(* Logix 5000 project; controller AdvManLab vendor 1 type 14 code 158 rev 28.12; software revision 28.01; part 4 of 13 *)
(* tags used below, declared in another part *)
   Inp : P_PF52x_Inp;   // Common part of PF523 / PF525 Input Assembly
   Out : P_PF52x_Out;   // Common part of PF523 / PF525 Output Assembly
   Inp_FwdPermOK : BOOL;   // 1=Permissives OK, drive can start Forward
   Inp_FwdNBPermOK : BOOL;   // 1=Non-Bypassable Permissives OK, drive can start Forward
   Inp_RevPermOK : BOOL;   // 1=Permissives OK, drive can start Reverse
   Inp_RevNBPermOK : BOOL;   // 1=Non-Bypassable Permissives OK, motor can start Reverse
   Inp_IntlkOK : BOOL;   // 1=Interlocks OK, drive can start/run
   Inp_NBIntlkOK : BOOL;   // 1=Non-Bypassable Interlocks OK, drive can start/run
   Inp_IOFault : BOOL;   // Input Communication Status 0=OK, 1=fail
   Inp_Sim : BOOL;   // 1=Simulate working drive; 0=Start/Stop/ Monitor actual drive
   Inp_Hand : BOOL;   // 1=Acquire Hand (typ. hardwired local) Mode, 0=Release Hand Mode
   Inp_OvrdCmd : SINT;   // Override Mode Command: 0=None, 1=Stop, 2=Start Fwd 3=Start Rev
   Inp_OvrdSpeed : REAL;   // Value to set Speed Reference in Override Mode (SpeedRef EU)
   Inp_Reset : BOOL;   // 1=Reset drive fault conditions and latched Alarms
   Cfg_HasReverse : BOOL;   // 1=Drive can be run reverse, 0=Forward only
   Cfg_AllowLocal : BOOL;   // 1=Allow Local Start/Stop without alarm, 0=Start/Stop from HMI/prog only
   Cfg_SetTrack : BOOL;   // 1=PSets track OSets in Oper, OSets track PSets in Prog, 0=no tracking
   Cfg_SetTrackOvrdHand : BOOL;   // 1=Prog/Oper Settings track Override/Hand speed reference
   Cfg_PCmdClear : ALIAS FOR Mode.Cfg_PCmdClear;
   Cfg_OCmdResets : BOOL;   // 1=New Oper drive cmd. resets fault, 0=reset req'd to clear fault
   Cfg_OvrdPermIntlk : BOOL;   // 1=Override ignores Bypassable Perm/ Intlk; 0=always use Perm/Intlk
   Cfg_ShedOnIOFault : BOOL;   // 1=Stop Motor and Alarm on I/O Fault; 0=Alarm only on I/O Fault
   Cfg_SimScaleEU : BOOL;   // 1=In simulation, scale Speed Ref EU to Speed Fdbk EU
   Cfg_SimScaleRaw : BOOL;   // 1=In simulation, scale Speed Ref EU to raw, then raw to Speed Fdbk EU
   Cfg_MinSpdRef : REAL;   // Minimum Speed Reference in EU (for limiting)
   Cfg_MaxSpdRef : REAL;   // Maximum Speed Reference in EU (for limiting)
   Cfg_SpeedRefRawMin : INT;   // Speed Reference Minimum in Drive (raw) Units (for scaling)
   Cfg_SpeedRefRawMax : INT;   // Speed Reference Maximum in Drive (raw) Units (for scaling)
   Cfg_SpeedRefEUMin : REAL;   // Speed Reference Minimum in Engineering Units (for scaling)
   Cfg_SpeedRefEUMax : REAL;   // Speed Reference Maximum in Engineering Units (for scaling)
   Cfg_SpeedFdbkRawMin : INT;   // Speed Feedback Minimum in Drive (raw) Units (for scaling)
   Cfg_SpeedFdbkRawMax : INT;   // Speed Feedback Maximum in Drive (raw) Units (for scaling)
   Cfg_SpeedFdbkEUMin : REAL;   // Speed Feedback Minimum in Engineering Units (for scaling)
   Cfg_SpeedFdbkEUMax : REAL;   // Speed Feedback Maximum in Engineering Units (for scaling)
   Cfg_SimRampT : DINT;   // Time to ramp speed fdbk when in Simulation (sec)
   Cfg_FailToStartT : DINT;   // Time after Start to get Run Feedback before Fault (sec)
   Cfg_FailToStopT : DINT;   // Time after Stop to drop Run Feedback before Fault (sec)
   Cfg_ResetPulseT : DINT;   // Time to pulse Out_Reset to clear drive fault
   Cfg_MaxJogT : REAL;   // Maximum jog time (sec, 0=unlimited)
   Cfg_OperKeep : SINT;   // Oper keeps control in Prog Mode: .0=Reference, .1=Start/Stop, .2=Fwd/Rev
   Cfg_ProgKeep : SINT;   // Prog keeps control in Oper Mode: .0=Reference, .1=Start/Stop, .2=Fwd/Rev
   PSet_SpeedRef : REAL;   // Program Setting of Speed Reference (EU)
   PSet_Owner : DINT;   // Program Owner Request ID (non-zero) or Release (zero)
   OSet_SpeedRef : REAL;   // Operator Setting of Speed Reference (EU)
   PCmd_Start : BOOL;   // Program Command to Start Drive
   PCmd_Fwd : BOOL;   // Program Command to set direction to Fowrard
   PCmd_Rev : BOOL;   // Program Command to set direction to Reverse
   PCmd_Reset : BOOL;   // Program Command to Reset drive fault and all Alarms requiring Reset
   PCmd_FailToStartAck : ALIAS FOR FailToStart.PCmd_Ack;   // Program Command to Acknowledge Fail to Start Alarm
   PCmd_FailToStopAck : ALIAS FOR FailToStop.PCmd_Ack;   // Program Command to Acknowledge Fail to Stop Alarm
   PCmd_IntlkTripAck : ALIAS FOR IntlkTrip.PCmd_Ack;   // Program Command to Acknowledge Interlock Trip Alarm
   PCmd_DriveFaultAck : ALIAS FOR DriveFault.PCmd_Ack;   // Program Command to Acknowledge Drive Fault Alarm
   PCmd_IOFaultAck : ALIAS FOR IOFault.PCmd_Ack;   // Program Command to Acknowledge I/O Fault Alarm
   OCmd_Start : BOOL;   // Operator Command to Start Drive
   OCmd_Stop : BOOL;   // Operator Command to Stop Drive
   OCmd_Jog : BOOL;   // Operator Command to Jog Drive (not cleared by P_PF52x!)
   OCmd_Fwd : BOOL;   // Operator Command to set direction to Forward
   OCmd_Rev : BOOL;   // Operator Command to set direction to Reverse
   OCmd_Bypass : BOOL;   // Operator Command to Bypass all Bypassable Interlocks and Permissives
   OCmd_Check : BOOL;   // Operator Command to Check (not bypass) all Interlocks and Permissives
   MCmd_Disable : BOOL;   // Maintenance Command to Disable Drive
   MCmd_Enable : BOOL;   // Maintenance Command to Enable (allow to run) Drive
   OCmd_Reset : BOOL;   // Operator Command to Reset all Alarms requiring Reset
   OCmd_ResetAckAll : BOOL;   // Operator Command to Reset all Alarms and latched Shed conditions
   Val_SpeedFdbk : REAL;   // Speed Feedback (actual) from drive
   Val_SpeedRefEUMin : REAL;   // Minimum of Speed Reference = MIN (Cfg_SpeedFdbkEUMin, Cfg_SpeedFdbkEUMax)
   Val_SpeedRefEUMax : REAL;   // Maximum of Speed Reference = MAX (Cfg_SpeedFdbkEUMin, Cfg_SpeedFdbkEUMax)
   Val_SpeedFdbkEUMin : REAL;   // Minimum of Speed Feedback = MIN (Cfg_SpeedFdbkEUMin, Cfg_SpeedFdbkEUMax)
   Val_SpeedFdbkEUMax : REAL;   // Maximum of Speed Feedback = MAX (Cfg_SpeedFdbkEUMin, Cfg_SpeedFdbkEUMax)
   Val_Fdbk : SINT;   // Device Feedback 0=Stopped, 1=Running Fwd 2=Running Rev 3=Accelerating 4=Decelerating
   Val_Owner : DINT;   // Current Object Owner ID (0=not owned)
   Sts_Starting : BOOL;   // 1=Drive requested to run and awaiting run feedback
   Sts_Running : BOOL;   // 1=Drive requested to run and is confirmed running
   Sts_CommandDir : BOOL;   // 1=Drive commanded to Forward, 0=Reverse
   Sts_ActualDir : BOOL;   // 1=Drive Actual direction is Forward, 0=Reverse
   Sts_Accel : BOOL;   // 1=Drive is Accelerating
   Sts_Decel : BOOL;   // 1=Drive is Decelerating
   Sts_NotReady : BOOL;   // 1=Device Not Ready, see detail bits for reason
   Sts_AtSpeed : BOOL;   // 1=Drive is running at reference speed
   Sts_Available : BOOL;   // 1=Drive available for control by automation (Prog)
   Sts_Bypass : BOOL;   // 1=Bypassable Interlocks and Permissives are Bypassed
   Sts_BypActive : BOOL;   // 1=Bypassing Active (Bypassed or Maintenance)
   Sts_Disabled : BOOL;   // 1=Drive is Disabled
   Sts_NotRdy : BOOL;   // 1=Motor is Not Ready to Run (independent of Mode)
   Nrdy_Disabled : BOOL;   // 1=Device Not Ready: Device Disabled by Maintenance
   Nrdy_CfgErr : BOOL;   // 1=Device Not Ready: Configuration Error
   Nrdy_Intlk : BOOL;   // 1=Device Not Ready: Interlock Not OK
   Nrdy_Perm : BOOL;   // 1=Device Not Ready: Permissive Not OK
   Nrdy_OperPrio : BOOL;   // 1=Device Not Ready: Operator State 0 Priority Command Requires Reset
   Nrdy_Fail : BOOL;   // 1=Device Not Ready: Device Failure (Shed Requires Reset)
   Nrdy_IOFault : BOOL;   // 1=Device Not Ready: I/O Fault (Shed Requires Reset)
   Nrdy_Trip : BOOL;   // 1=Device not Ready: Deivce Tripped (Drive Fault)
   Nrdy_DriveNR : BOOL;   // 1=Device Note Ready: Drive Not Ready
   Nrdy_NoMode : BOOL;   // 1=Device Not Ready: Device Logic Disabled / NO Mode
   Sts_MaintByp : BOOL;   // 1=A Maintenance Bypass is Active, display icon
   Sts_Err : BOOL;   // 1=Error in Config: see detail bits for reason
   Err_Timer : BOOL;   // 1=Error in Config: Invalid Check or Reset Pulse Time (use 0 to 2147483)
   Err_Sim : BOOL;   // 1=Error in Config: simulation timer preset: use 0 to 2147483)
   Err_Alarm : BOOL;   // 1=Error in Config: Alarm Min On Time, Shelf Time, Severity
   Err_FdbkRaw : BOOL;   // 1=Erron in Config: Speed Fdbk Raw Min = Max
   Err_FdbkEU : BOOL;   // 1=Error in Config: Speed Fdbk EU Min = Max
   Err_RefLim : BOOL;   // 1=Error in Config: Speed Ref Limit Min > Max
   Err_RefEU : BOOL;   // 1=Error in Config: Speed Ref EU Min = Max
   Err_RefRaw : BOOL;   // 1=Error in Config: Speed Ref Raw Min = Max
   Sts_Hand : ALIAS FOR Mode.Sts_Hand;
   Sts_Maint : ALIAS FOR Mode.Sts_Maint;
   Sts_Ovrd : ALIAS FOR Mode.Sts_Ovrd;
   Sts_Prog : ALIAS FOR Mode.Sts_Prog;
   Sts_Oper : ALIAS FOR Mode.Sts_Oper;
   Sts_FailToStart : ALIAS FOR FailToStart.Inp;   // 1=Drive Failed to Start (One-Shot)
   Sts_FailToStop : ALIAS FOR FailToStop.Inp;   // 1=Drive Failed to Stop
   Sts_IntlkTrip : ALIAS FOR IntlkTrip.Inp;   // 1=Drive was stopped by an Interlock NOT OK (One-Shot)
   Sts_DriveFault : ALIAS FOR DriveFault.Inp;   // 1=Drive Fault (see drive display or manual)
   Sts_IOFault : ALIAS FOR IOFault.Inp;   // I/O Comm Fault Status (0=OK, 1=Bad)
   Rdy_Fwd : BOOL;   // 1=Ready to receive OCmd_Fwd (enabled HMI button)
   Rdy_Rev : BOOL;   // 1=Ready to receive OCmd_Rev (enables HMI button)
   Rdy_Bypass : BOOL;   // 1=Ready to receive OCmd_Bypass (enables HMI button)
   Rdy_Check : BOOL;   // 1=Ready to receive OCmd_Check (enables HMI button)
   Rdy_Disable : BOOL;   // 1=Ready to receive MCmd_Disable (enables HMI button)
   Rdy_Enable : BOOL;   // 1=Ready to receive MCmd_Enable (enables HMI button)
   Rdy_SpeedRef : BOOL;   // 1=Ready to receive OSet_SpeedRef (enables data entry field)
   P_PF52x : BOOL;   // Unique Parameter Name for auto - discovery
   Mode : P_Mode;   // Drive Mode Selection
   IOFault : P_Alarm;   // I/O Fault Alarm
   IntlkTrip : P_Alarm;   // Interlock Trip Alarm
   FailToStop : P_Alarm;   // Drive Failed to Stop Alarm
   FailToStart : P_Alarm;   // Drive Failed to Start Alarm
   Cfg_Tag : STRING_20;   // Tagname for display on HMI
   Cfg_Label : STRING_20;   // Label for graphic symbol displayed on HMI
   Cfg_Desc : STRING_40;   // Description for display on HMI
   Wrk_Run : BOOL;   // 1=Drive should be "running", 0=should be "stopped"
   Wrk_StartRetrigT : TIMER;   // Time to pulse start output on start command retrigger (Maint)
   Wrk_StopRetrigT : TIMER;   // Time to pulse stop output on stop command retrigger (Maint)
   Wrk_RunFdbk : BOOL;   // Run Feedback based on mode, simulation, etc. 1=running
   Wrk_Bypass : BOOL;   // Internal Bypassable Permissives and Interlocks are Bypassed flag
   Wrk_Disabled : BOOL;   // Internal Drive is Disabled
   DriveFault : P_Alarm;   // Drive Faulted Alarm
   Cfg_SpeedRefEU : STRING_8;   // Speed Reference Engineering Units for display on HMI
   Wrk_SpeedRef : REAL;   // Working copy of Speed Reference (for limiting)
   Wrk_Rev : BOOL;   // Working (internal) Direction 1=Reverse 0=Forward (default)
   Wrk_Jog : BOOL;   // 1=Jog Drive, 0=Drive not jogging
   Wrk_ResetT : TIMER;   // Reset Output Pulse Timer
   Wrk_ResetONS : BOOL;   // One-Shot to fire Reset Timer to ensure min. output ON time.
   Cfg_SpeedFdbkEU : STRING_8;   // Speed Feedback Engineering Units for display on HMI
   Cfg_RevText : STRING_16;   // Name for Reverse Direction, e.g., "Down", "Reverse"
   Cfg_FwdText : STRING_16;   // Name for Forward Direction, e.g., "Up", "Forward"
   Wrk_StopT : TIMER;   // Stop Check Timer (for Fail to Stop)
   Wrk_StartT : TIMER;   // Start Check Timer (for Fail to Start)
   Wrk_Retrigger : BOOL;   // Maint Start issued while running or Stop while stopped
   Wrk_Step : REAL;   // Amount to change simulated Speed Fdbk this scan (ramp)
   Wrk_ScanTime : REAL;   // Seconds since previous scan
   Wrk_ScanT : TIMER;   // Scan Timer (milliseconds, always runs)
   Wrk_SimFdbkTgt : REAL;   // Speed Ref converted to Speed Fdbk units for simulation: target speed fdbk
   Inf_Type : STRING_16;   // Type identifier for HMI navigation
   Wrk_JogT : TIMER;   // Jog Timer
   Val_FaultDesc : STRING_40;   // Description of Drive Fault (given LastFaultCode)
   Wrk_ProgKeep2ONS : BOOL;   // Prog Keep bit 2 one-shot store
   Wrk_ProgKeep1ONS : BOOL;   // Prog Keep bit 1 one-shot store
   Wrk_ProgKeep0ONS : BOOL;   // Prog Keep bit 0 one-shot store
   Wrk_OperKeep2ONS : BOOL;   // Oper Keep bit 2 one-shot store
   Wrk_OperKeep1ONS : BOOL;   // Oper Keep bit 1 one-shot store
   Wrk_OperKeep0ONS : BOOL;   // Oper Keep bit 0 one-shot store
   Inf_Lib : STRING_12;   // Display Library for Faceplate call-up
   Cfg_DigIn4Txt : STRING_20;   // Drive Digital Input 4 Label
   Cfg_DigIn3Txt : STRING_20;   // Drive Digital Input 3 Label
   Cfg_DigIn2Txt : STRING_20;   // Drive Digital Input 2 Label
   Cfg_DigIn1Txt : STRING_20;   // Drive Digital Input 1 Label
   ONS : DINT;
   Running : BOOL;
(* P_PF52x, continued *)

ROUTINE Logic   (* ladder *)
// Normal Scan: control / monitor Variable-Speed Drive
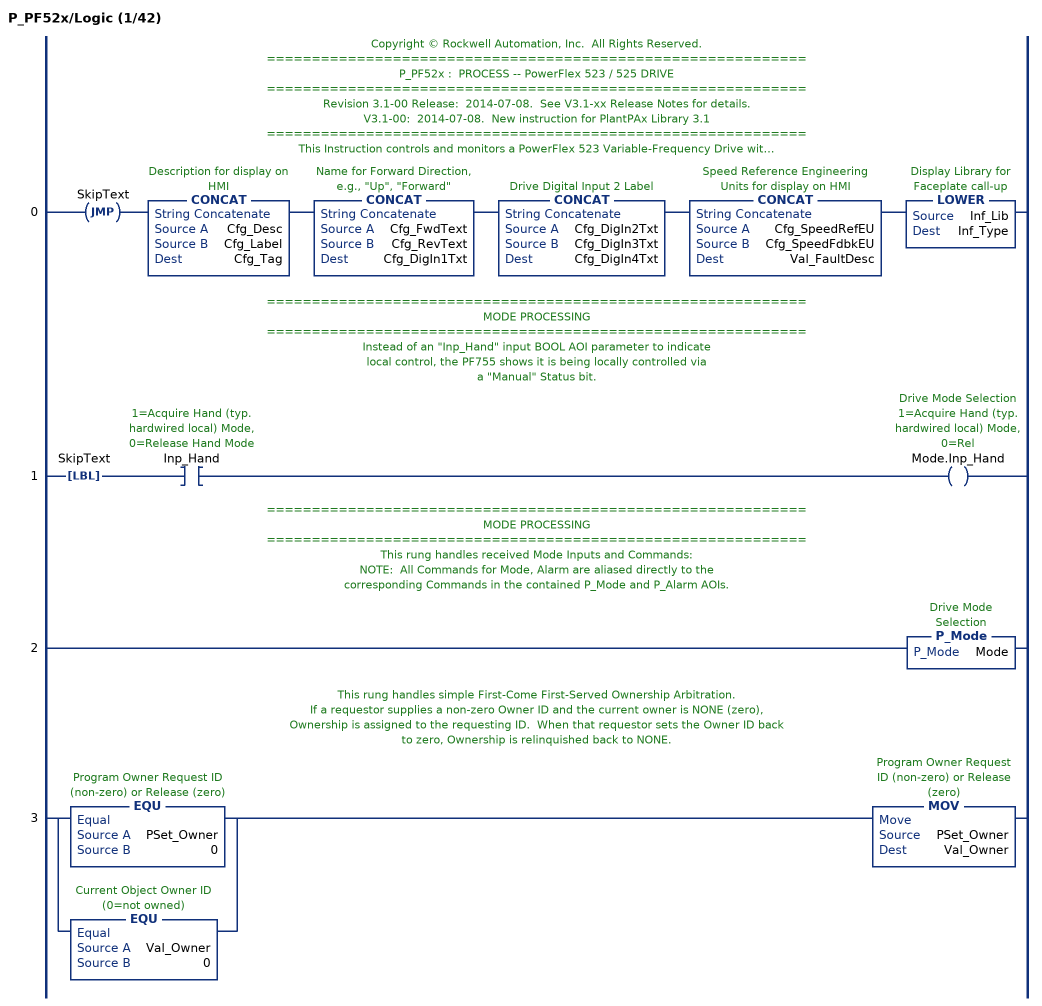
   // Copyright © Rockwell Automation, Inc.  All Rights Reserved.
   // ============================================================
   // P_PF52x :  PROCESS -- PowerFlex 523 / 525 DRIVE
   // ============================================================
   // Revision 3.1-00 Release:  2014-07-08.  See V3.1-xx Release Notes for details.
   // V3.1-00:  2014-07-08.  New instruction for PlantPAx Library 3.1
   // ============================================================
   // This Instruction controls and monitors a PowerFlex 523 Variable-Frequency Drive with
   // optional EtherNet/IP Interface, or a PowerFlex 525 Variable-Frequency
   // Drive with embedded or optional add-on EtherNet/IP Interface.
   // This instruction provides:
   // *  Starting, stopping, jogging of drive, setting speed reference and direction
   // *  Monitoring of run feedback, display of actual drive status, including accel, decel, direction, speed
   // *  Detection of Failure to Start, Failure to Stop, Drive Fault
   // *  Monitoring of Permissive conditions to allow starting
   // * Monitoring of Interlock conditions to stop / prevent starting
   // * Simulation, providing feedback of a working drive while disabling outputs
   // * Monitoring of I/O communication faults
   // * Alarms for Fail to Start, Fail to Stop, Interlock Trip, Drive Fault, I/O Fault
   // * Option to automatically reset faults and alarms when operator commands
   // motor to start or stop
   // * Supports HMI "breadcrumbs" for Alarm Inhibited, Bad Configuration,
   // Not Ready, Maintenance Bypass Active
   // * "Available" status for use by automation logic to know whether motor
   // can be controlled by other objects.
   // Modes are provided by a P_Mode Add-On Instruction instance.
   // Alarms are provided by P_Alarm Add-On Instruction instances.
   // Modes of operation: Operator, Program, Override, Maintenance, Hand
   // See Rockwell Automation Publication 520COM-UM001_ for information on
   // the PowerFlex 525 embedded EtherNet/IP interface.
   // See Rockwell Automation Publication 520COM-UM003_ for information on
   // the PowerFlex 525 add-on EtherNet/IP interface (dual-port).
   // See Rockwell Automation Publication 520-UM001_ for information on the
   // PowerFlex 523 and 525 drive parameters and programming
   // ============================================================
   // SHOW LOCAL STRINGS
   // ============================================================
   // The STRINGs containing the text associated with each instance of this
   // instruction cannot be Input or Output Parameters, because STRINGs are not
   //  'atomic' types. (Inputs and Outputs must be SINT, INT, DINT, REAL, or BOOL.)
   // In order to make it easier to find and configure these STRINGs, this rung
   // was added.  THE JMP (and the LBL on the following rung)
   // MUST NOT BE REMOVED!!!
   // To view the STRINGs, go to the instruction instance (in LD or FBD), RIGHT-click
   // to bring up the context menu and select "Open Instruction Logic".
   // This rung will appear with the STRING values for the selected instance.
   // You may double-click the STRING values here to modify them as well.
   0: JMP(SkipText)CONCAT(Cfg_Desc,Cfg_Label,Cfg_Tag)CONCAT(Cfg_FwdText,Cfg_RevText,Cfg_DigIn1Txt)CONCAT(Cfg_DigIn2Txt,Cfg_DigIn3Txt,Cfg_DigIn4Txt)CONCAT(Cfg_SpeedRefEU,Cfg_SpeedFdbkEU,Val_FaultDesc)LOWER(Inf_Lib,Inf_Type);
   // ============================================================
   // MODE PROCESSING
   // ============================================================
   // Instead of an "Inp_Hand" input BOOL AOI parameter to indicate
   // local control, the PF755 shows it is being locally controlled via
   // a "Manual" Status bit.
   1: LBL(SkipText)XIC(Inp_Hand)OTE(Mode.Inp_Hand);
   // ============================================================
   // MODE PROCESSING
   // ============================================================
   // This rung handles received Mode Inputs and Commands:
   // NOTE:  All Commands for Mode, Alarm are aliased directly to the
   // corresponding Commands in the contained P_Mode and P_Alarm AOIs.
   2: P_Mode(Mode);
   // This rung handles simple First-Come First-Served Ownership Arbitration.
   // If a requestor supplies a non-zero Owner ID and the current owner is NONE (zero),
   // Ownership is assigned to the requesting ID.  When that requestor sets the Owner ID back
   // to zero, Ownership is relinquished back to NONE.
   3: [EQU(PSet_Owner,0) ,EQU(Val_Owner,0) ]MOV(PSet_Owner,Val_Owner);
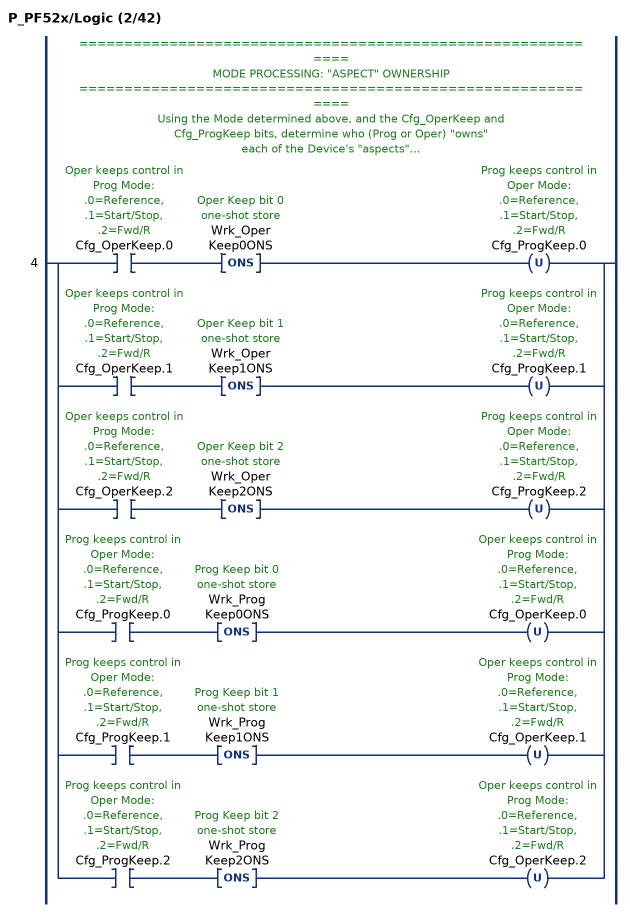
   // ============================================================
   // MODE PROCESSING: "ASPECT" OWNERSHIP
   // ============================================================
   // Using the Mode determined above, and the Cfg_OperKeep and
   // Cfg_ProgKeep bits, determine who (Prog or Oper) "owns"
   // each of the Device's "aspects":
   // Speed Reference (.0), Start/Stop (.1),
   // and Forward/Reverse (.2).
   // The bits within Cfg_OperKeep and Cfg_ProgKeep determine which "aspects"
   // (sub-functions of this AOI) are retained by the Operator in Program Mode,
   // or by the Program in Operator Mode (respectively).
   // All aspects (functions) may be "kept" (basically locking the Operator/Program Mode
   // selection, rendering it moot --  you get to explain how it works to your operators!!!),
   // but it is NOT allowed to have any given function retained by BOTH Operator and
   // Program.  This rung ensures that no function is "kept" by both Oper and Prog.
   4: [XIC(Cfg_OperKeep.0) ONS(Wrk_OperKeep0ONS) OTU(Cfg_ProgKeep.0) ,XIC(Cfg_OperKeep.1) ONS(Wrk_OperKeep1ONS) OTU(Cfg_ProgKeep.1) ,XIC(Cfg_OperKeep.2) ONS(Wrk_OperKeep2ONS) OTU(Cfg_ProgKeep.2) ,XIC(Cfg_ProgKeep.0) ONS(Wrk_ProgKeep0ONS) OTU(Cfg_OperKeep.0) ,XIC(Cfg_ProgKeep.1) ONS(Wrk_ProgKeep1ONS) OTU(Cfg_OperKeep.1) ,XIC(Cfg_ProgKeep.2) ONS(Wrk_ProgKeep2ONS) OTU(Cfg_OperKeep.2) ];
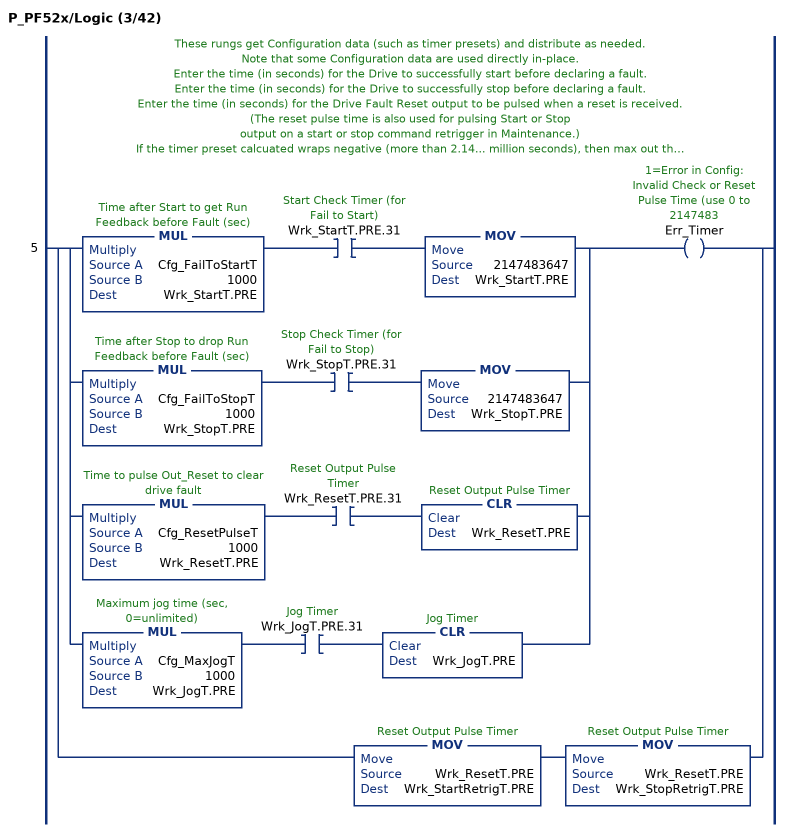
   // These rungs get Configuration data (such as timer presets) and distribute as needed.
   // Note that some Configuration data are used directly in-place.
   // Enter the time (in seconds) for the Drive to successfully start before declaring a fault.
   // Enter the time (in seconds) for the Drive to successfully stop before declaring a fault.
   // Enter the time (in seconds) for the Drive Fault Reset output to be pulsed when a reset is received.
   // (The reset pulse time is also used for pulsing Start or Stop
   // output on a start or stop command retrigger in Maintenance.)
   // If the timer preset calcuated wraps negative (more than 2.14... million seconds), then max out the
   // or clear the Timer Preset (as appropriate) and flag it.  Note that a negative timer preset will fault the controller!!!
   5: [[MUL(Cfg_FailToStartT,1000,Wrk_StartT.PRE) XIC(Wrk_StartT.PRE.31) MOV(2147483647,Wrk_StartT.PRE) ,MUL(Cfg_FailToStopT,1000,Wrk_StopT.PRE) XIC(Wrk_StopT.PRE.31) MOV(2147483647,Wrk_StopT.PRE) ,MUL(Cfg_ResetPulseT,1000,Wrk_ResetT.PRE) XIC(Wrk_ResetT.PRE.31) CLR(Wrk_ResetT.PRE) ,MUL(Cfg_MaxJogT,1000,Wrk_JogT.PRE) XIC(Wrk_JogT.PRE.31) CLR(Wrk_JogT.PRE) ] OTE(Err_Timer) ,MOV(Wrk_ResetT.PRE,Wrk_StartRetrigT.PRE) MOV(Wrk_ResetT.PRE,Wrk_StopRetrigT.PRE) ];
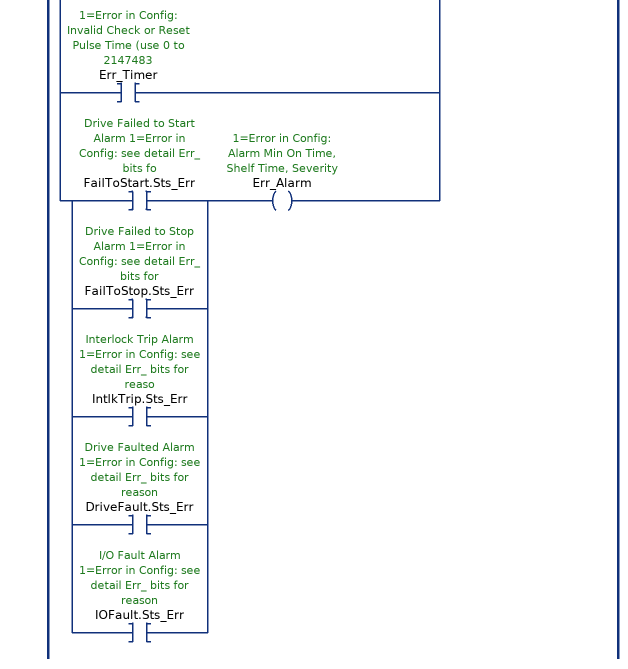
   // This rung handles the reports of all Bad Configuration Status.
   // Individual bits are provided for various status:
   // Bad Raw Scaling configs
   // Bad Engineering Units Scaling configs
   // Bad Min or Max Speed Reference clamp limit
   // Bad simulation speed ramp time
   // Bad timer config from (rung above)
   // Bad Alarm config (from P_Alarm)
   // Bad Cfg_OperKeep / Cfg_ProgKeep config
   // Then a summary Bad Config status is provided, simply an OR of the individual bits.
   6: [EQU(Cfg_SpeedFdbkRawMax,Cfg_SpeedFdbkRawMin) OTE(Err_FdbkRaw) ,EQU(Cfg_SpeedFdbkEUMax,Cfg_SpeedFdbkEUMin) OTE(Err_FdbkEU) ,EQU(Cfg_SpeedRefEUMax,Cfg_SpeedRefEUMin) OTE(Err_RefEU) ,EQU(Cfg_SpeedRefRawMax,Cfg_SpeedRefRawMin) OTE(Err_RefRaw) ,[LEQ(Cfg_MaxSpdRef,Cfg_MinSpdRef) ,LES(Cfg_MinSpdRef,0.0) ] OTE(Err_RefLim) ,LES(Cfg_SimRampT,0) OTE(Err_Sim) ,XIC(Err_Timer) ,[XIC(FailToStart.Sts_Err) ,XIC(FailToStop.Sts_Err) ,XIC(IntlkTrip.Sts_Err) ,XIC(DriveFault.Sts_Err) ,XIC(IOFault.Sts_Err) ] OTE(Err_Alarm) ]OTE(Sts_Err);
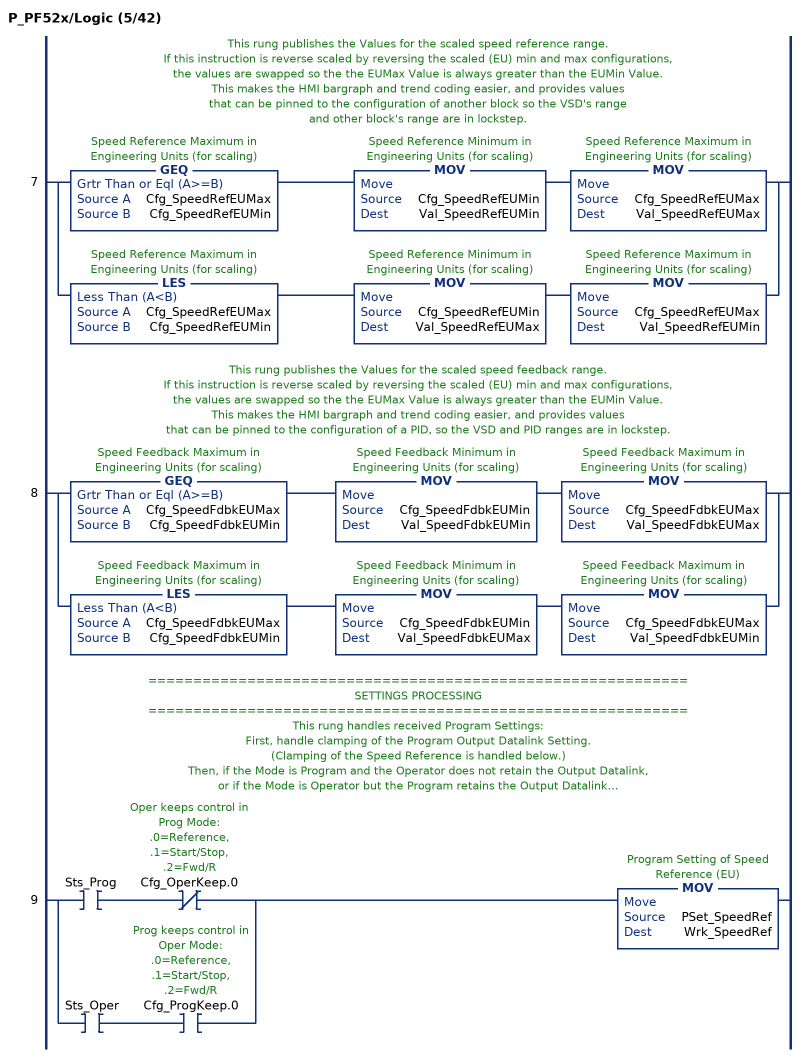
   // This rung publishes the Values for the scaled speed reference range.
   // If this instruction is reverse scaled by reversing the scaled (EU) min and max configurations,
   // the values are swapped so the the EUMax Value is always greater than the EUMin Value.
   // This makes the HMI bargraph and trend coding easier, and provides values
   // that can be pinned to the configuration of another block so the VSD's range
   //  and other block's range are in lockstep.
   7: [GEQ(Cfg_SpeedRefEUMax,Cfg_SpeedRefEUMin) MOV(Cfg_SpeedRefEUMin,Val_SpeedRefEUMin) MOV(Cfg_SpeedRefEUMax,Val_SpeedRefEUMax) ,LES(Cfg_SpeedRefEUMax,Cfg_SpeedRefEUMin) MOV(Cfg_SpeedRefEUMin,Val_SpeedRefEUMax) MOV(Cfg_SpeedRefEUMax,Val_SpeedRefEUMin) ];
   // This rung publishes the Values for the scaled speed feedback range.
   // If this instruction is reverse scaled by reversing the scaled (EU) min and max configurations,
   // the values are swapped so the the EUMax Value is always greater than the EUMin Value.
   // This makes the HMI bargraph and trend coding easier, and provides values
   // that can be pinned to the configuration of a PID, so the VSD and PID ranges are in lockstep.
   8: [GEQ(Cfg_SpeedFdbkEUMax,Cfg_SpeedFdbkEUMin) MOV(Cfg_SpeedFdbkEUMin,Val_SpeedFdbkEUMin) MOV(Cfg_SpeedFdbkEUMax,Val_SpeedFdbkEUMax) ,LES(Cfg_SpeedFdbkEUMax,Cfg_SpeedFdbkEUMin) MOV(Cfg_SpeedFdbkEUMin,Val_SpeedFdbkEUMax) MOV(Cfg_SpeedFdbkEUMax,Val_SpeedFdbkEUMin) ];
   // ============================================================
   // SETTINGS PROCESSING
   // ============================================================
   // This rung handles received Program Settings:
   // First, handle clamping of the Program Output Datalink Setting.
   // (Clamping of the Speed Reference is handled below.)
   // Then, if the Mode is Program and the Operator does not retain the Output Datalink,
   // or if the Mode is Operator but the Program retains the Output Datalink,
   // use the Program Setting for the Output Datalink.
   // The Program Setting for the Speed Reference is handled similarly.
   9: [XIC(Sts_Prog) XIO(Cfg_OperKeep.0) ,XIC(Sts_Oper) XIC(Cfg_ProgKeep.0) ]MOV(PSet_SpeedRef,Wrk_SpeedRef);
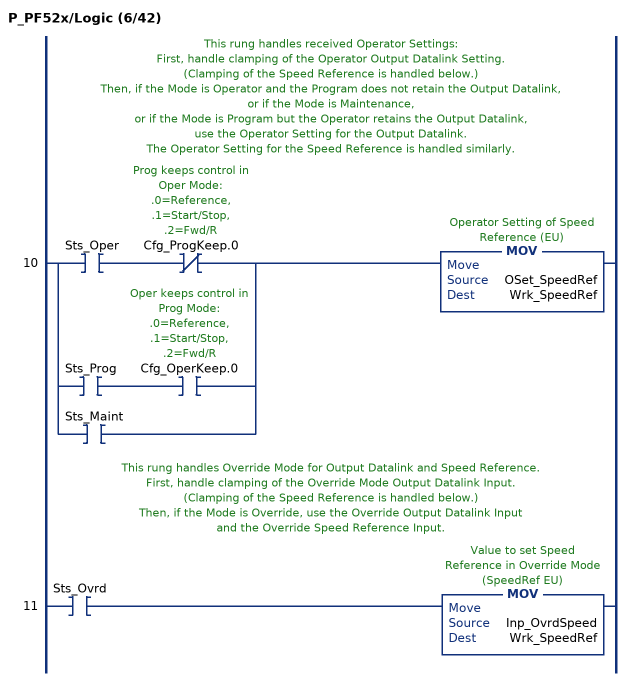
   // This rung handles received Operator Settings:
   // First, handle clamping of the Operator Output Datalink Setting.
   // (Clamping of the Speed Reference is handled below.)
   // Then, if the Mode is Operator and the Program does not retain the Output Datalink,
   // or if the Mode is Maintenance,
   // or if the Mode is Program but the Operator retains the Output Datalink,
   // use the Operator Setting for the Output Datalink.
   // The Operator Setting for the Speed Reference is handled similarly.
   10: [XIC(Sts_Oper) XIO(Cfg_ProgKeep.0) ,XIC(Sts_Prog) XIC(Cfg_OperKeep.0) ,XIC(Sts_Maint) ]MOV(OSet_SpeedRef,Wrk_SpeedRef);
   // This rung handles Override Mode for Output Datalink and Speed Reference.
   // First, handle clamping of the Override Mode Output Datalink Input.
   // (Clamping of the Speed Reference is handled below.)
   // Then, if the Mode is Override, use the Override Output Datalink Input
   // and the Override Speed Reference Input.
   11: XIC(Sts_Ovrd)MOV(Inp_OvrdSpeed,Wrk_SpeedRef);
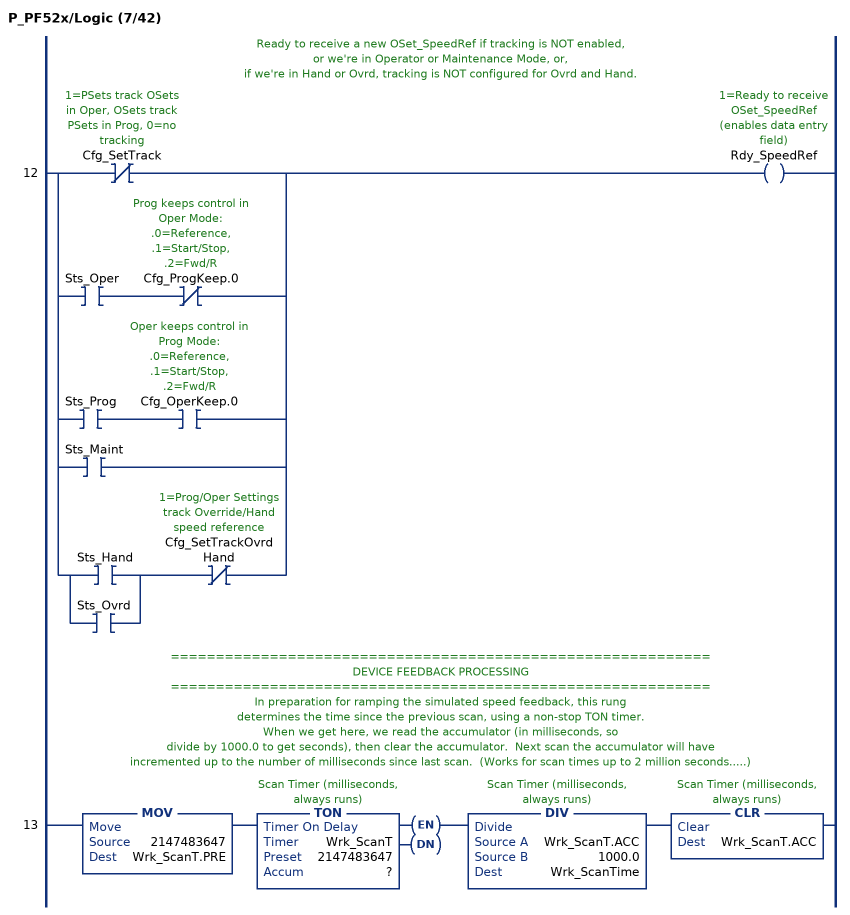
   // Ready to receive a new OSet_SpeedRef if tracking is NOT enabled,
   // or we're in Operator or Maintenance Mode, or,
   // if we're in Hand or Ovrd, tracking is NOT configured for Ovrd and Hand.
   12: [XIO(Cfg_SetTrack) ,XIC(Sts_Oper) XIO(Cfg_ProgKeep.0) ,XIC(Sts_Prog) XIC(Cfg_OperKeep.0) ,XIC(Sts_Maint) ,[XIC(Sts_Hand) ,XIC(Sts_Ovrd) ] XIO(Cfg_SetTrackOvrdHand) ]OTE(Rdy_SpeedRef);
   // ============================================================
   // DEVICE FEEDBACK PROCESSING
   // ============================================================
   // In preparation for ramping the simulated speed feedback, this rung
   // determines the time since the previous scan, using a non-stop TON timer.
   // When we get here, we read the accumulator (in milliseconds, so
   // divide by 1000.0 to get seconds), then clear the accumulator.  Next scan the accumulator will have
   // incremented up to the number of milliseconds since last scan.  (Works for scan times up to 2 million seconds.....)
   13: MOV(2147483647,Wrk_ScanT.PRE)TON(Wrk_ScanT,?,?)DIV(Wrk_ScanT.ACC,1000.0,Wrk_ScanTime)CLR(Wrk_ScanT.ACC);
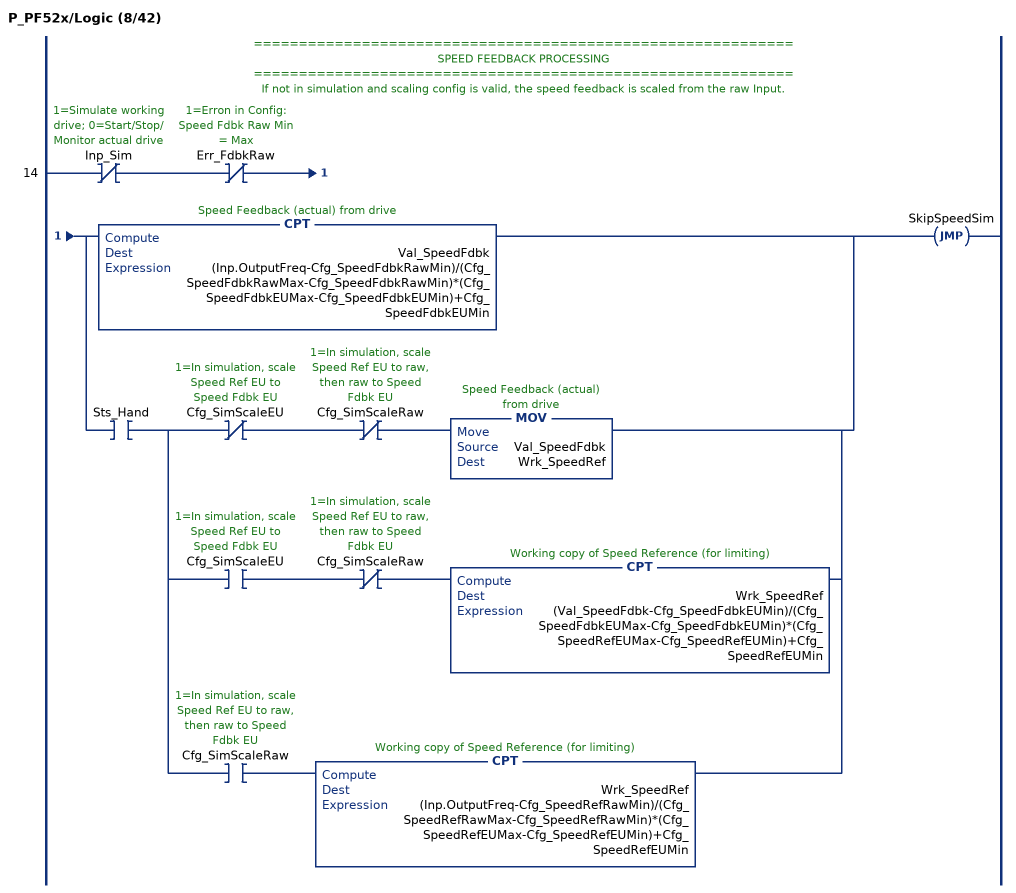
   // ============================================================
   // SPEED FEEDBACK PROCESSING
   // ============================================================
   // If not in simulation and scaling config is valid, the speed feedback is scaled from the raw Input.
   14: XIO(Inp_Sim)XIO(Err_FdbkRaw)[CPT(Val_SpeedFdbk,(Inp.OutputFreq-Cfg_SpeedFdbkRawMin)/(Cfg_SpeedFdbkRawMax-Cfg_SpeedFdbkRawMin)*(Cfg_SpeedFdbkEUMax-Cfg_SpeedFdbkEUMin)+Cfg_SpeedFdbkEUMin) ,XIC(Sts_Hand) [XIO(Cfg_SimScaleEU) XIO(Cfg_SimScaleRaw) MOV(Val_SpeedFdbk,Wrk_SpeedRef) ,[XIC(Cfg_SimScaleEU) XIO(Cfg_SimScaleRaw) CPT(Wrk_SpeedRef,(Val_SpeedFdbk-Cfg_SpeedFdbkEUMin)/(Cfg_SpeedFdbkEUMax-Cfg_SpeedFdbkEUMin)*(Cfg_SpeedRefEUMax-Cfg_SpeedRefEUMin)+Cfg_SpeedRefEUMin) ,XIC(Cfg_SimScaleRaw) CPT(Wrk_SpeedRef,(Inp.OutputFreq-Cfg_SpeedRefRawMin)/(Cfg_SpeedRefRawMax-Cfg_SpeedRefRawMin)*(Cfg_SpeedRefEUMax-Cfg_SpeedRefEUMin)+Cfg_SpeedRefEUMin) ] ] ]JMP(SkipSpeedSim);
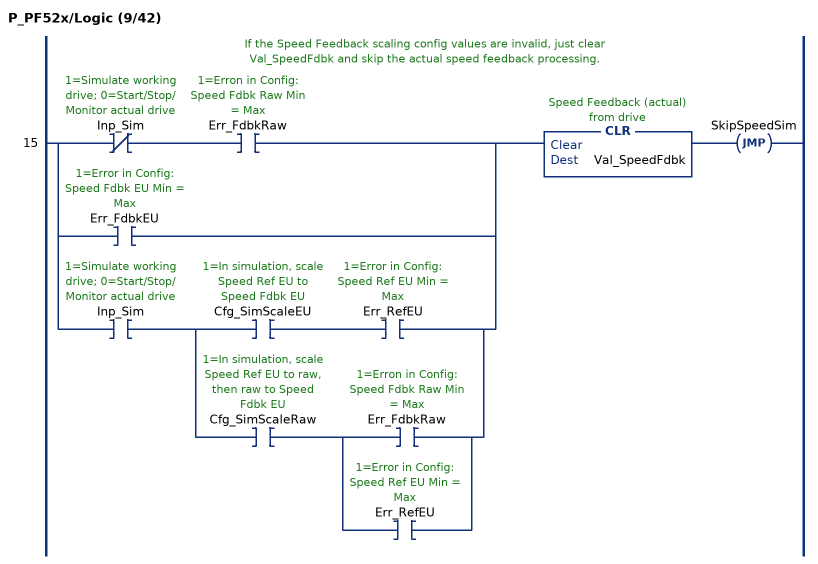
   // If the Speed Feedback scaling config values are invalid, just clear
   // Val_SpeedFdbk and skip the actual speed feedback processing.
   15: [XIO(Inp_Sim) XIC(Err_FdbkRaw) ,XIC(Err_FdbkEU) ,XIC(Inp_Sim) [XIC(Cfg_SimScaleEU) XIC(Err_RefEU) ,XIC(Cfg_SimScaleRaw) [XIC(Err_FdbkRaw) ,XIC(Err_RefEU) ] ] ]CLR(Val_SpeedFdbk)JMP(SkipSpeedSim);
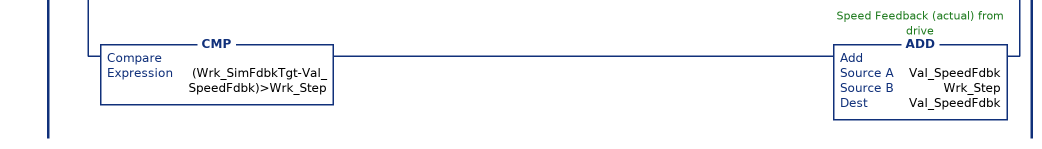
   // If in simulation, simulate accel/decel.
   16: XIC(Inp_Sim)[[XIC(Wrk_Run) ,XIC(Wrk_Jog) ] [XIO(Cfg_SimScaleEU) XIO(Cfg_SimScaleRaw) MOV(Wrk_SpeedRef,Wrk_SimFdbkTgt) ,[XIC(Cfg_SimScaleEU) XIO(Cfg_SimScaleRaw) CPT(Wrk_SimFdbkTgt,(Wrk_SpeedRef-Cfg_SpeedRefEUMin)/(Cfg_SpeedRefEUMax-Cfg_SpeedRefEUMin)*(Cfg_SpeedFdbkEUMax-Cfg_SpeedFdbkEUMin)+Cfg_SpeedFdbkEUMin) ,XIC(Cfg_SimScaleRaw) [CPT(Wrk_SimFdbkTgt,(Wrk_SpeedRef-Cfg_SpeedRefEUMin)/(Cfg_SpeedRefEUMax-Cfg_SpeedRefEUMin)*(Cfg_SpeedRefRawMax-Cfg_SpeedRefRawMin)+Cfg_SpeedRefRawMin) ,CPT(Wrk_SimFdbkTgt,(Wrk_SimFdbkTgt-Cfg_SpeedFdbkRawMin)/(Cfg_SpeedFdbkRawMax-Cfg_SpeedFdbkRawMin)*(Cfg_SpeedFdbkEUMax-Cfg_SpeedFdbkEUMin)+Cfg_SpeedFdbkEUMin) ] ] ] ,[XIO(Wrk_Run) XIO(Wrk_Jog) ,XIO(Wrk_Rev) XIO(Sts_ActualDir) ,XIC(Wrk_Rev) XIC(Sts_ActualDir) ] CLR(Wrk_SimFdbkTgt) ,GRT(Cfg_SimRampT,0) [CPT(Wrk_Step,Cfg_MaxSpdRef/Cfg_SimRampT*Wrk_ScanTime) ,XIC(Cfg_SimScaleEU) XIO(Cfg_SimScaleRaw) CPT(Wrk_Step,(Wrk_Step-Cfg_SpeedRefEUMin)/(Cfg_SpeedRefEUMax-Cfg_SpeedRefEUMin)*(Cfg_SpeedFdbkEUMax-Cfg_SpeedFdbkEUMin)+Cfg_SpeedFdbkEUMin) ,XIC(Cfg_SimScaleRaw) [CPT(Wrk_Step,(Wrk_Step-Cfg_SpeedRefEUMin)/(Cfg_SpeedRefEUMax-Cfg_SpeedRefEUMin)*(Cfg_SpeedRefRawMax-Cfg_SpeedRefRawMin)+Cfg_SpeedRefRawMin) ,CPT(Wrk_Step,(Wrk_Step-Cfg_SpeedFdbkRawMin)/(Cfg_SpeedFdbkRawMax-Cfg_SpeedFdbkRawMin)*(Cfg_SpeedFdbkEUMax-Cfg_SpeedFdbkEUMin)+Cfg_SpeedFdbkEUMin) ] ] ,LEQ(Cfg_SimRampT,0) MOV(1.50000000e+038,Wrk_Step) ,CMP(ABS(Val_SpeedFdbk-Wrk_SimFdbkTgt)<=Wrk_Step) MOV(Wrk_SimFdbkTgt,Val_SpeedFdbk) ,CMP((Val_SpeedFdbk-Wrk_SimFdbkTgt)>Wrk_Step) SUB(Val_SpeedFdbk,Wrk_Step,Val_SpeedFdbk) ,CMP((Wrk_SimFdbkTgt-Val_SpeedFdbk)>Wrk_Step) ADD(Val_SpeedFdbk,Wrk_Step,Val_SpeedFdbk) ];
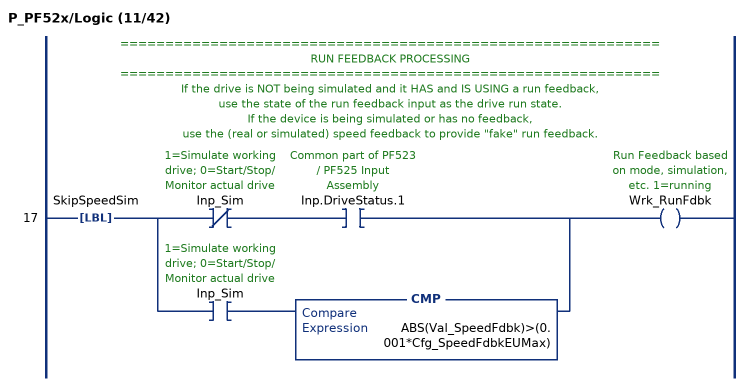
   // ============================================================
   // RUN FEEDBACK PROCESSING
   // ============================================================
   // If the drive is NOT being simulated and it HAS and IS USING a run feedback,
   // use the state of the run feedback input as the drive run state.
   // If the device is being simulated or has no feedback,
   // use the (real or simulated) speed feedback to provide "fake" run feedback.
   17: LBL(SkipSpeedSim)[XIO(Inp_Sim) XIC(Inp.DriveStatus.1) ,XIC(Inp_Sim) CMP(ABS(Val_SpeedFdbk)>(0.001*Cfg_SpeedFdbkEUMax)) ]OTE(Wrk_RunFdbk);
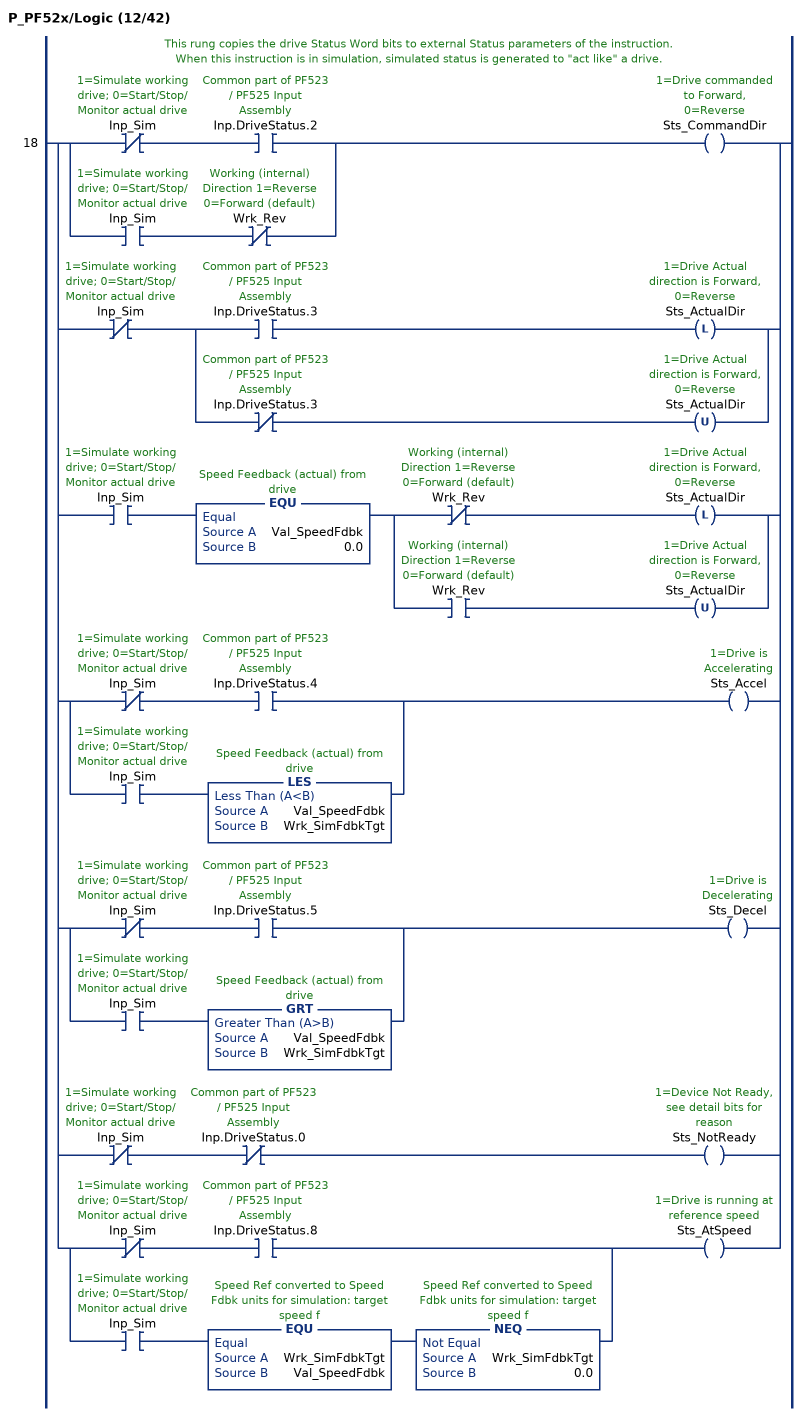
   // This rung copies the drive Status Word bits to external Status parameters of the instruction.
   // When this instruction is in simulation, simulated status is generated to "act like" a drive.
   18: [[XIO(Inp_Sim) XIC(Inp.DriveStatus.2) ,XIC(Inp_Sim) XIO(Wrk_Rev) ] OTE(Sts_CommandDir) ,[XIO(Inp_Sim) [XIC(Inp.DriveStatus.3) OTL(Sts_ActualDir) ,XIO(Inp.DriveStatus.3) OTU(Sts_ActualDir) ] ,XIC(Inp_Sim) EQU(Val_SpeedFdbk,0.0) [XIO(Wrk_Rev) OTL(Sts_ActualDir) ,XIC(Wrk_Rev) OTU(Sts_ActualDir) ] ] ,[XIO(Inp_Sim) XIC(Inp.DriveStatus.4) ,XIC(Inp_Sim) LES(Val_SpeedFdbk,Wrk_SimFdbkTgt) ] OTE(Sts_Accel) ,[XIO(Inp_Sim) XIC(Inp.DriveStatus.5) ,XIC(Inp_Sim) GRT(Val_SpeedFdbk,Wrk_SimFdbkTgt) ] OTE(Sts_Decel) ,XIO(Inp_Sim) XIO(Inp.DriveStatus.0) OTE(Sts_NotReady) ,[XIO(Inp_Sim) XIC(Inp.DriveStatus.8) ,XIC(Inp_Sim) EQU(Wrk_SimFdbkTgt,Val_SpeedFdbk) NEQ(Wrk_SimFdbkTgt,0.0) ] OTE(Sts_AtSpeed) ];
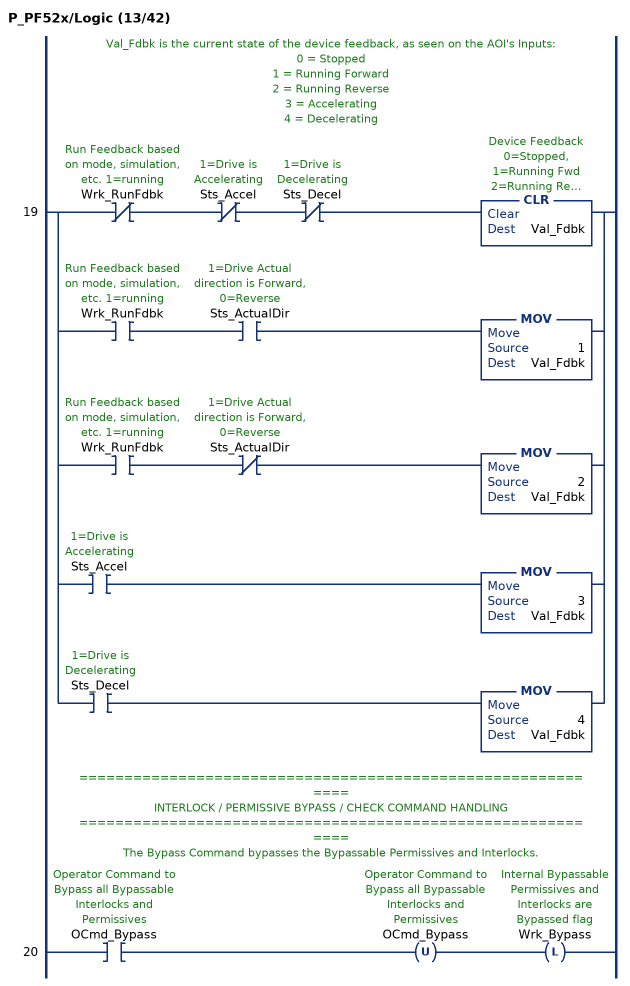
   // Val_Fdbk is the current state of the device feedback, as seen on the AOI's Inputs:
   // 0 = Stopped
   // 1 = Running Forward
   // 2 = Running Reverse
   // 3 = Accelerating
   // 4 = Decelerating
   19: [XIO(Wrk_RunFdbk) XIO(Sts_Accel) XIO(Sts_Decel) CLR(Val_Fdbk) ,XIC(Wrk_RunFdbk) XIC(Sts_ActualDir) MOV(1,Val_Fdbk) ,XIC(Wrk_RunFdbk) XIO(Sts_ActualDir) MOV(2,Val_Fdbk) ,XIC(Sts_Accel) MOV(3,Val_Fdbk) ,XIC(Sts_Decel) MOV(4,Val_Fdbk) ];
   // ============================================================
   // INTERLOCK / PERMISSIVE BYPASS / CHECK COMMAND HANDLING
   // ============================================================
   // The Bypass Command bypasses the Bypassable Permissives and Interlocks.
   20: XIC(OCmd_Bypass)OTU(OCmd_Bypass)OTL(Wrk_Bypass);
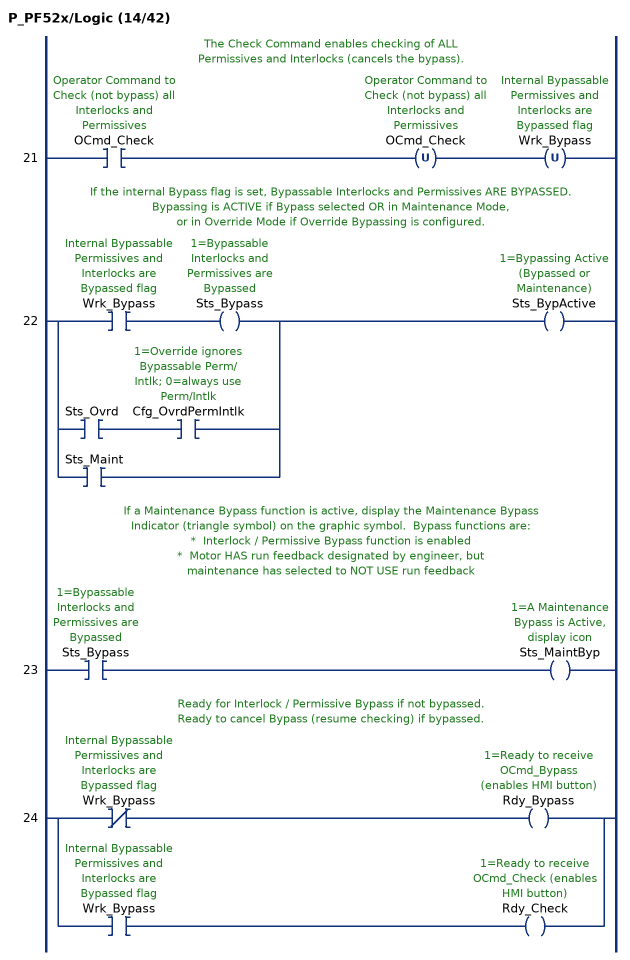
   // The Check Command enables checking of ALL
   // Permissives and Interlocks (cancels the bypass).
   21: XIC(OCmd_Check)OTU(OCmd_Check)OTU(Wrk_Bypass);
   // If the internal Bypass flag is set, Bypassable Interlocks and Permissives ARE BYPASSED.
   // Bypassing is ACTIVE if Bypass selected OR in Maintenance Mode,
   // or in Override Mode if Override Bypassing is configured.
   22: [XIC(Wrk_Bypass) OTE(Sts_Bypass) ,XIC(Sts_Ovrd) XIC(Cfg_OvrdPermIntlk) ,XIC(Sts_Maint) ]OTE(Sts_BypActive);
   // If a Maintenance Bypass function is active, display the Maintenance Bypass
   // Indicator (triangle symbol) on the graphic symbol.  Bypass functions are:
   // *  Interlock / Permissive Bypass function is enabled
   // *  Motor HAS run feedback designated by engineer, but
   // maintenance has selected to NOT USE run feedback
   23: XIC(Sts_Bypass)OTE(Sts_MaintByp);
   // Ready for Interlock / Permissive Bypass if not bypassed.
   // Ready to cancel Bypass (resume checking) if bypassed.
   24: [XIO(Wrk_Bypass) OTE(Rdy_Bypass) ,XIC(Wrk_Bypass) OTE(Rdy_Check) ];
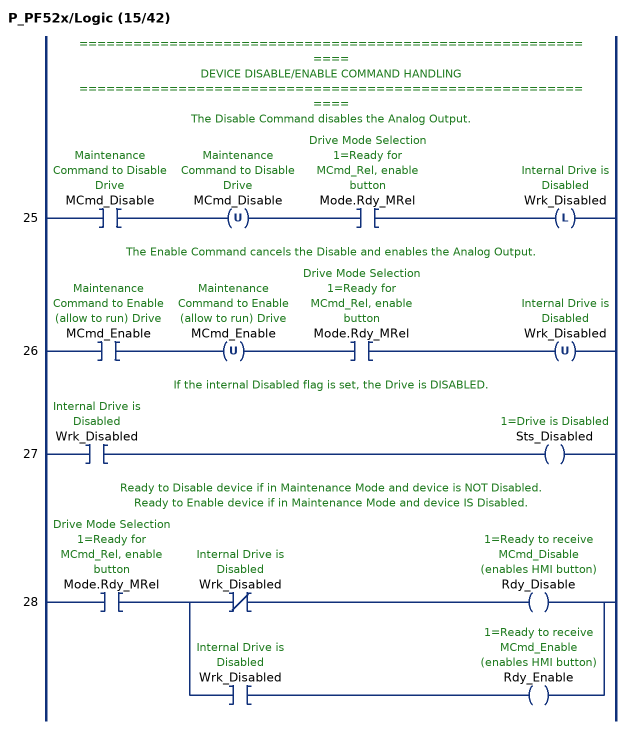
   // ============================================================
   // DEVICE DISABLE/ENABLE COMMAND HANDLING
   // ============================================================
   // The Disable Command disables the Analog Output.
   25: XIC(MCmd_Disable)OTU(MCmd_Disable)XIC(Mode.Rdy_MRel)OTL(Wrk_Disabled);
   // The Enable Command cancels the Disable and enables the Analog Output.
   26: XIC(MCmd_Enable)OTU(MCmd_Enable)XIC(Mode.Rdy_MRel)OTU(Wrk_Disabled);
   // If the internal Disabled flag is set, the Drive is DISABLED.
   27: XIC(Wrk_Disabled)OTE(Sts_Disabled);
   // Ready to Disable device if in Maintenance Mode and device is NOT Disabled.
   // Ready to Enable device if in Maintenance Mode and device IS Disabled.
   28: XIC(Mode.Rdy_MRel)[XIO(Wrk_Disabled) OTE(Rdy_Disable) ,XIC(Wrk_Disabled) OTE(Rdy_Enable) ];
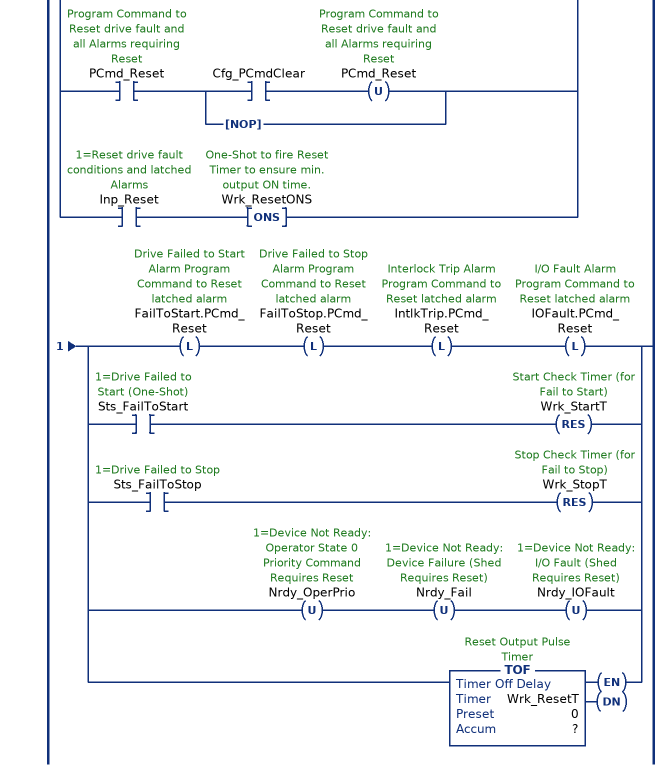
   // ============================================================
   // ALARM RESET COMMAND HANDLING
   // ============================================================
   // This rung handles the Alarm Reset Input and Commands
   // and the "Reset and Ack All" Operator Command.
   // This rung processes received Reset Commands from:
   // 1.  The Operator via HMI Operator Command, or
   // 2.  Higher-level strategies via Program Command
   // 3.  Pushbuttons or other block via Input
   // 4.  Resets initiated by other device Operator Commands (if configured to do so)
   // and forwards the Reset to ALL Alarms and latched Shed conditions.
   // The reset starts the Reset Timer (One-Shot Off-Delay)
   // to ensure the output is held on for at least the minimum time.
   29: [[XIC(OCmd_Reset) OTU(OCmd_Reset) ,[XIC(OCmd_Start) ,XIC(OCmd_Stop) ] XIC(Cfg_OCmdResets) [XIC(Sts_Oper) XIO(Cfg_ProgKeep.1) ,XIC(Sts_Prog) XIC(Cfg_OperKeep.1) ,XIC(Sts_Maint) ] ] ,XIC(OCmd_ResetAckAll) OTU(OCmd_ResetAckAll) [OTL(PCmd_FailToStartAck) ,OTL(PCmd_FailToStopAck) ,OTL(PCmd_DriveFaultAck) ,OTL(PCmd_IntlkTripAck) ,OTL(PCmd_IOFaultAck) ] ,XIC(PCmd_Reset) [XIC(Cfg_PCmdClear) OTU(PCmd_Reset) ,NOP() ] ,XIC(Inp_Reset) ONS(Wrk_ResetONS) ][OTL(FailToStart.PCmd_Reset) OTL(FailToStop.PCmd_Reset) OTL(IntlkTrip.PCmd_Reset) OTL(IOFault.PCmd_Reset) ,XIC(Sts_FailToStart) RES(Wrk_StartT) ,XIC(Sts_FailToStop) RES(Wrk_StopT) ,OTU(Nrdy_OperPrio) OTU(Nrdy_Fail) OTU(Nrdy_IOFault) ,TOF(Wrk_ResetT,?,?) ];
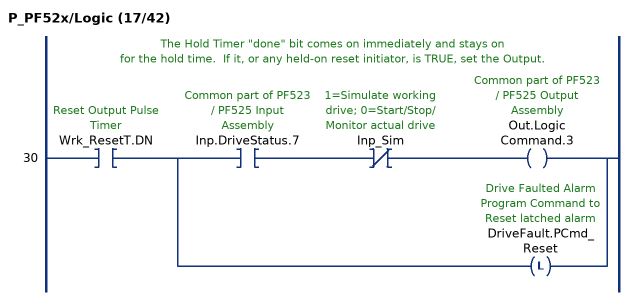
   // The Hold Timer "done" bit comes on immediately and stays on
   // for the hold time.  If it, or any held-on reset initiator, is TRUE, set the Output.
   30: XIC(Wrk_ResetT.DN)[XIC(Inp.DriveStatus.7) XIO(Inp_Sim) OTE(Out.LogicCommand.3) ,OTL(DriveFault.PCmd_Reset) ];
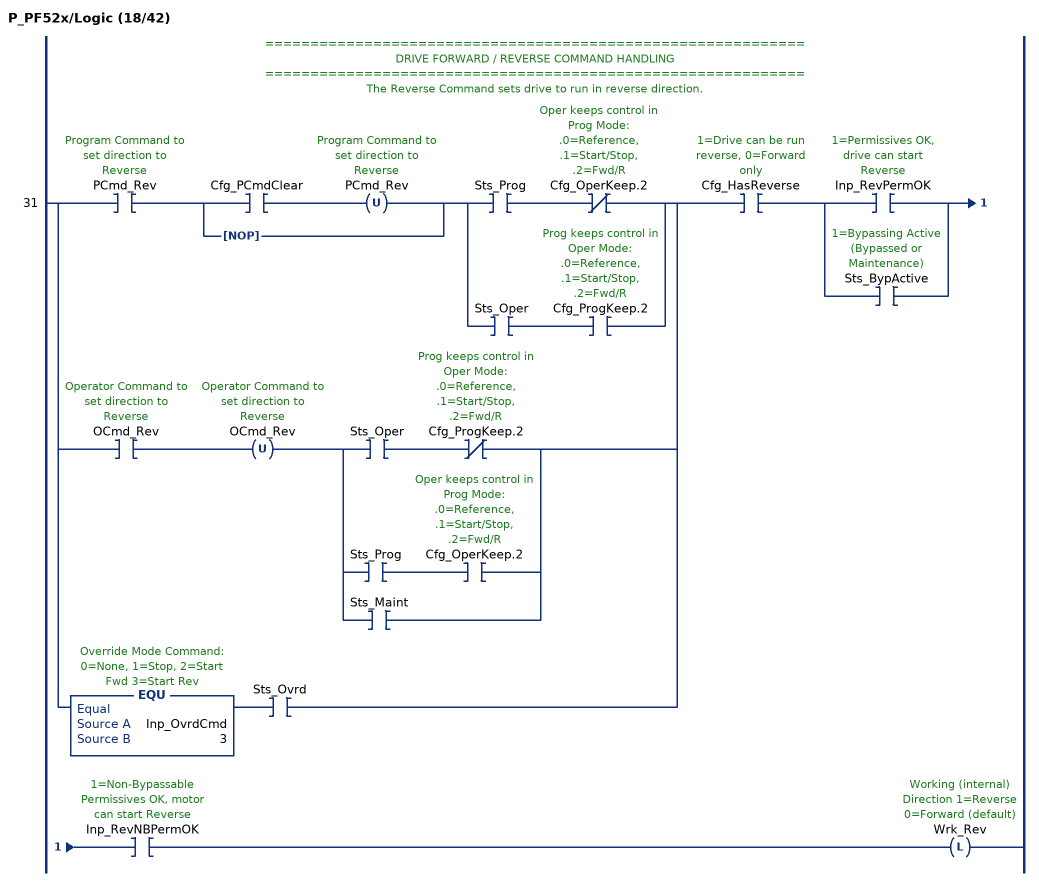
   // ============================================================
   // DRIVE FORWARD / REVERSE COMMAND HANDLING
   // ============================================================
   // The Reverse Command sets drive to run in reverse direction.
   31: [XIC(PCmd_Rev) [XIC(Cfg_PCmdClear) OTU(PCmd_Rev) ,NOP() ] [XIC(Sts_Prog) XIO(Cfg_OperKeep.2) ,XIC(Sts_Oper) XIC(Cfg_ProgKeep.2) ] ,XIC(OCmd_Rev) OTU(OCmd_Rev) [XIC(Sts_Oper) XIO(Cfg_ProgKeep.2) ,XIC(Sts_Prog) XIC(Cfg_OperKeep.2) ,XIC(Sts_Maint) ] ,EQU(Inp_OvrdCmd,3) XIC(Sts_Ovrd) ]XIC(Cfg_HasReverse)[XIC(Inp_RevPermOK) ,XIC(Sts_BypActive) ]XIC(Inp_RevNBPermOK)OTL(Wrk_Rev);
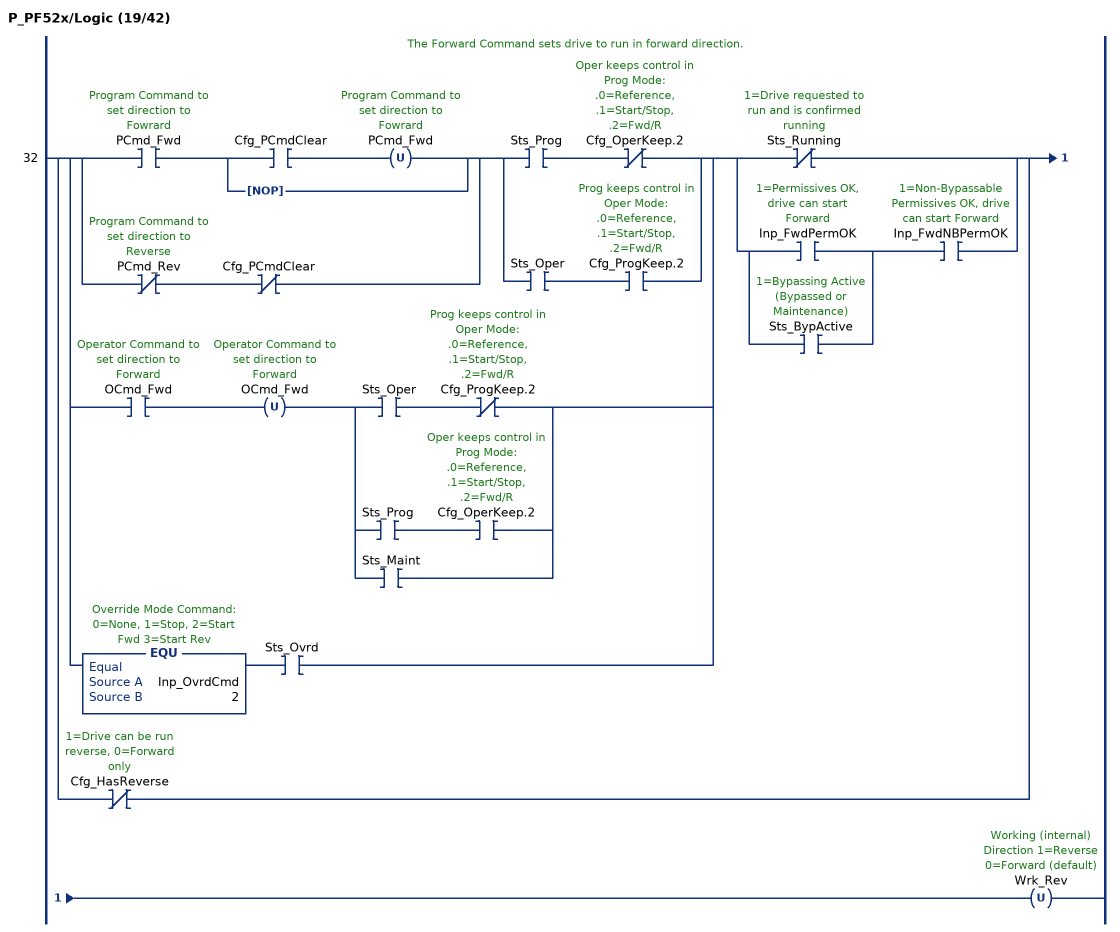
   // The Forward Command sets drive to run in forward direction.
   32: [[[XIC(PCmd_Fwd) [XIC(Cfg_PCmdClear) OTU(PCmd_Fwd) ,NOP() ] ,XIO(PCmd_Rev) XIO(Cfg_PCmdClear) ] [XIC(Sts_Prog) XIO(Cfg_OperKeep.2) ,XIC(Sts_Oper) XIC(Cfg_ProgKeep.2) ] ,XIC(OCmd_Fwd) OTU(OCmd_Fwd) [XIC(Sts_Oper) XIO(Cfg_ProgKeep.2) ,XIC(Sts_Prog) XIC(Cfg_OperKeep.2) ,XIC(Sts_Maint) ] ,EQU(Inp_OvrdCmd,2) XIC(Sts_Ovrd) ] [XIO(Sts_Running) ,[XIC(Inp_FwdPermOK) ,XIC(Sts_BypActive) ] XIC(Inp_FwdNBPermOK) ] ,XIO(Cfg_HasReverse) ]OTU(Wrk_Rev);
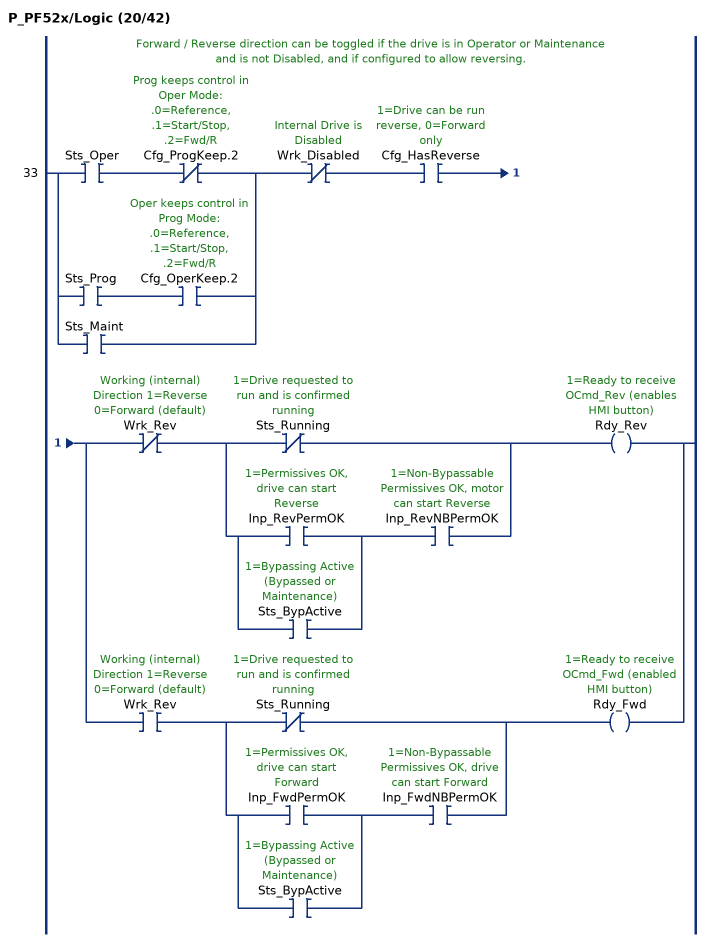
   // Forward / Reverse direction can be toggled if the drive is in Operator or Maintenance
   // and is not Disabled, and if configured to allow reversing.
   33: [XIC(Sts_Oper) XIO(Cfg_ProgKeep.2) ,XIC(Sts_Prog) XIC(Cfg_OperKeep.2) ,XIC(Sts_Maint) ]XIO(Wrk_Disabled)XIC(Cfg_HasReverse)[XIO(Wrk_Rev) [XIO(Sts_Running) ,[XIC(Inp_RevPermOK) ,XIC(Sts_BypActive) ] XIC(Inp_RevNBPermOK) ] OTE(Rdy_Rev) ,XIC(Wrk_Rev) [XIO(Sts_Running) ,[XIC(Inp_FwdPermOK) ,XIC(Sts_BypActive) ] XIC(Inp_FwdNBPermOK) ] OTE(Rdy_Fwd) ];
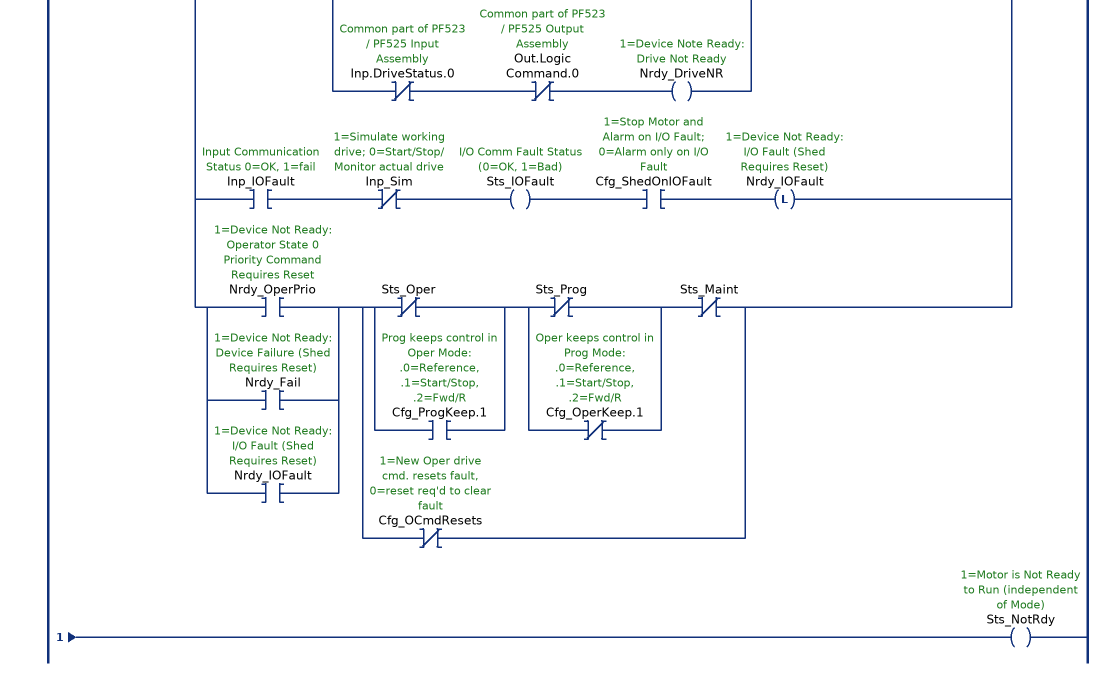
   // ============================================================
   // DRIVE START / STOP COMMAND HANDLING
   // ============================================================
   // The drive is NOT READY TO RUN if:
   // * Interlocks are not OK and not bypassed;
   // * Non-bypassable Interlocks are not OK;
   // * Permissives are not OK and not bypassed,
   // or Non-Bypassable Permissives are not OK,
   // and the motor is not already starting or running;
   // * The drive (not simulated) reports that it is faulted;
   // * There's an I/O failure and the motor is NOT being simulated;
   // * The motor has a Fail to Start that has not been reset;
   // * The drive is disabled (by Maintenance);
   // * This instruction instance has a configuration error.
   34: OTU(Nrdy_NoMode)[XIC(Sts_Disabled) OTE(Nrdy_Disabled) ,XIC(Sts_Err) OTE(Nrdy_CfgErr) ,[XIO(Inp_IntlkOK) XIO(Sts_BypActive) ,XIO(Inp_NBIntlkOK) ] [[XIC(Wrk_Run) ,XIC(Wrk_Jog) ] OTE(Sts_IntlkTrip) ,OTE(Nrdy_Intlk) ] ,[[XIO(Inp_FwdPermOK) XIO(Sts_BypActive) ,XIO(Inp_FwdNBPermOK) ] XIO(Wrk_Rev) ,[XIO(Inp_RevPermOK) XIO(Sts_BypActive) ,XIO(Inp_RevNBPermOK) ] XIC(Wrk_Rev) ] XIO(Sts_Starting) XIO(Sts_Running) OTE(Nrdy_Perm) ,XIO(Inp_Sim) [XIC(Inp.DriveStatus.7) OTE(Sts_DriveFault) OTE(Nrdy_Trip) ,XIO(Inp.DriveStatus.0) XIO(Out.LogicCommand.0) OTE(Nrdy_DriveNR) ] ,XIC(Inp_IOFault) XIO(Inp_Sim) OTE(Sts_IOFault) XIC(Cfg_ShedOnIOFault) OTL(Nrdy_IOFault) ,[XIC(Nrdy_OperPrio) ,XIC(Nrdy_Fail) ,XIC(Nrdy_IOFault) ] [[XIO(Sts_Oper) ,XIC(Cfg_ProgKeep.1) ] [XIO(Sts_Prog) ,XIO(Cfg_OperKeep.1) ] XIO(Sts_Maint) ,XIO(Cfg_OCmdResets) ] ]OTE(Sts_NotRdy);
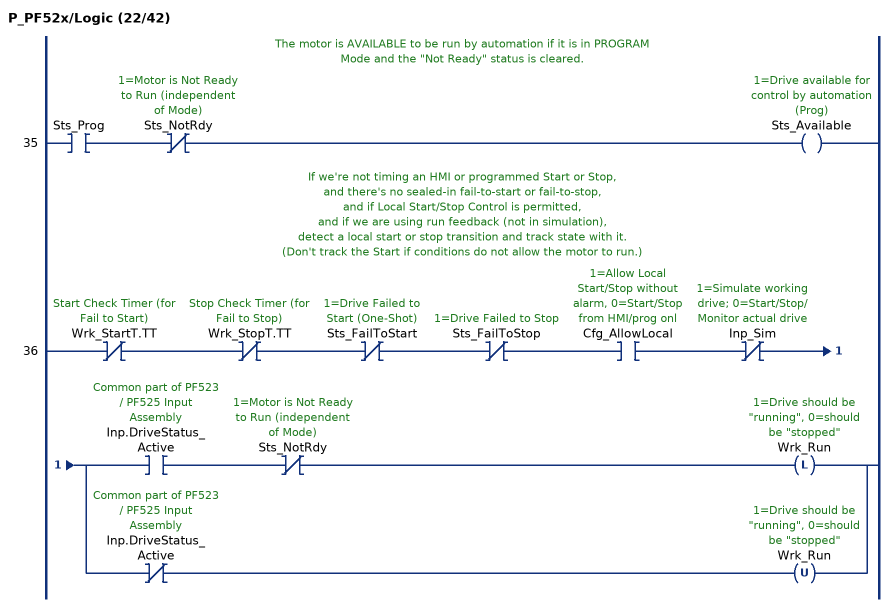
   // The motor is AVAILABLE to be run by automation if it is in PROGRAM
   // Mode and the "Not Ready" status is cleared.
   35: XIC(Sts_Prog)XIO(Sts_NotRdy)OTE(Sts_Available);
   // If we're not timing an HMI or programmed Start or Stop,
   // and there's no sealed-in fail-to-start or fail-to-stop,
   // and if Local Start/Stop Control is permitted,
   // and if we are using run feedback (not in simulation),
   // detect a local start or stop transition and track state with it.
   // (Don't track the Start if conditions do not allow the motor to run.)
   36: XIO(Wrk_StartT.TT)XIO(Wrk_StopT.TT)XIO(Sts_FailToStart)XIO(Sts_FailToStop)XIC(Cfg_AllowLocal)XIO(Inp_Sim)[XIC(Inp.DriveStatus_Active) XIO(Sts_NotRdy) OTL(Wrk_Run) ,XIO(Inp.DriveStatus_Active) OTU(Wrk_Run) ];
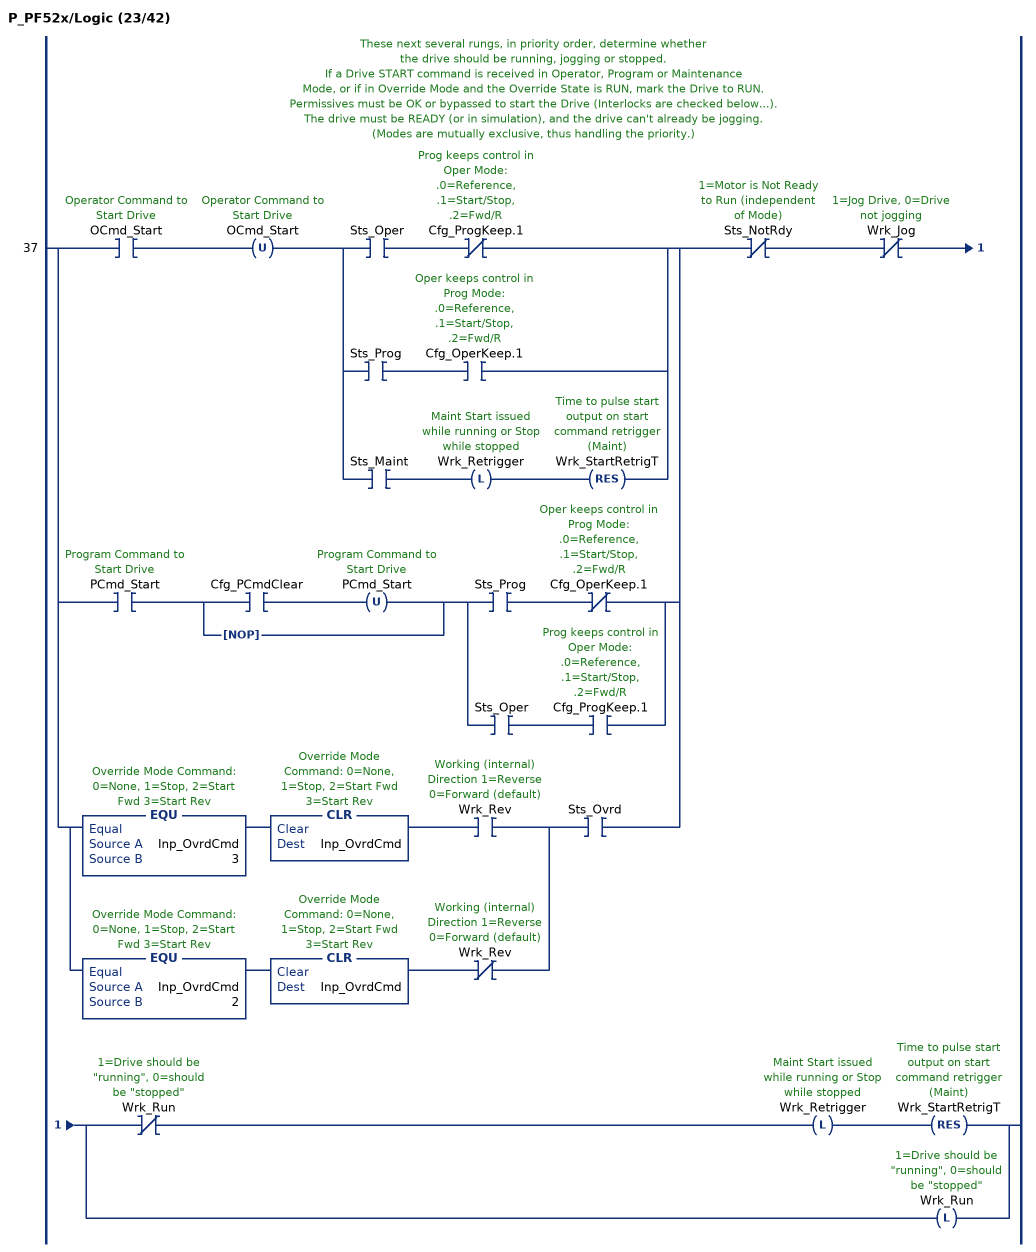
   // These next several rungs, in priority order, determine whether
   // the drive should be running, jogging or stopped.
   // If a Drive START command is received in Operator, Program or Maintenance
   // Mode, or if in Override Mode and the Override State is RUN, mark the Drive to RUN.
   // Permissives must be OK or bypassed to start the Drive (Interlocks are checked below...).
   // The drive must be READY (or in simulation), and the drive can't already be jogging.
   // (Modes are mutually exclusive, thus handling the priority.)
   37: [XIC(OCmd_Start) OTU(OCmd_Start) [XIC(Sts_Oper) XIO(Cfg_ProgKeep.1) ,XIC(Sts_Prog) XIC(Cfg_OperKeep.1) ,XIC(Sts_Maint) OTL(Wrk_Retrigger) RES(Wrk_StartRetrigT) ] ,XIC(PCmd_Start) [XIC(Cfg_PCmdClear) OTU(PCmd_Start) ,NOP() ] [XIC(Sts_Prog) XIO(Cfg_OperKeep.1) ,XIC(Sts_Oper) XIC(Cfg_ProgKeep.1) ] ,[EQU(Inp_OvrdCmd,3) CLR(Inp_OvrdCmd) XIC(Wrk_Rev) ,EQU(Inp_OvrdCmd,2) CLR(Inp_OvrdCmd) XIO(Wrk_Rev) ] XIC(Sts_Ovrd) ]XIO(Sts_NotRdy)XIO(Wrk_Jog)[XIO(Wrk_Run) OTL(Wrk_Retrigger) RES(Wrk_StartRetrigT) ,OTL(Wrk_Run) ];
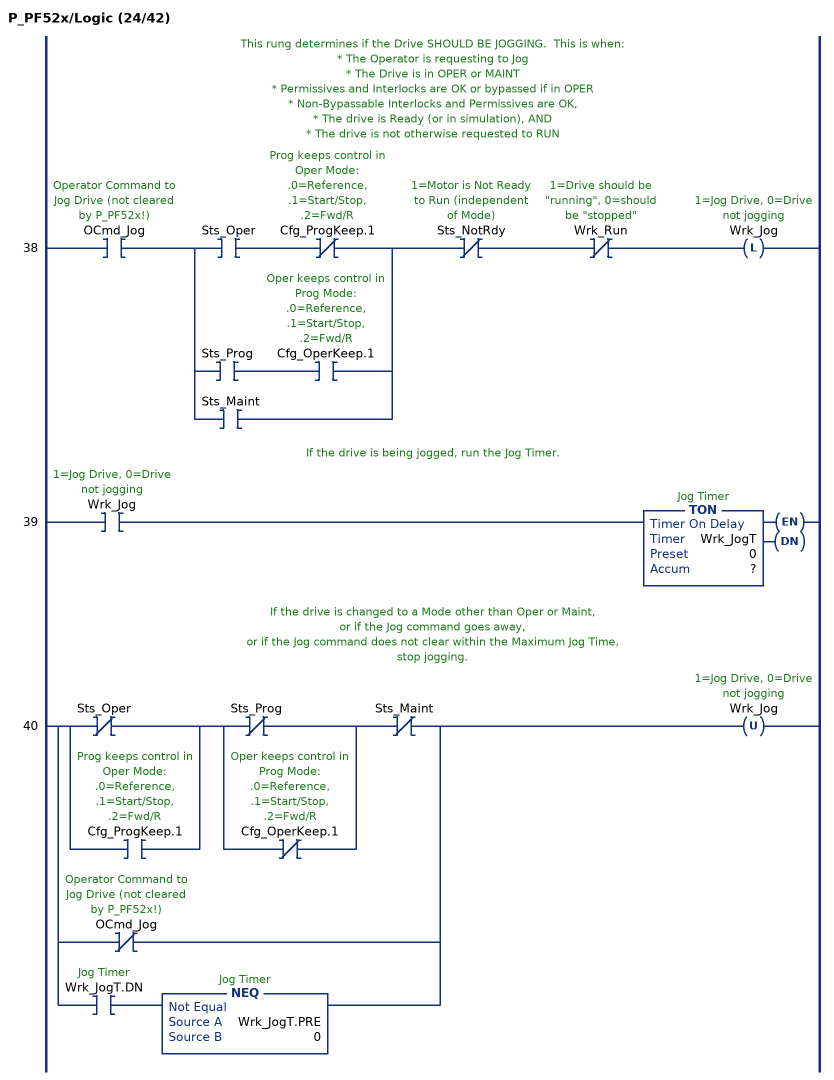
   // This rung determines if the Drive SHOULD BE JOGGING.  This is when:
   // * The Operator is requesting to Jog
   // * The Drive is in OPER or MAINT
   // * Permissives and Interlocks are OK or bypassed if in OPER
   // * Non-Bypassable Interlocks and Permissives are OK,
   // * The drive is Ready (or in simulation), AND
   // * The drive is not otherwise requested to RUN
   38: XIC(OCmd_Jog)[XIC(Sts_Oper) XIO(Cfg_ProgKeep.1) ,XIC(Sts_Prog) XIC(Cfg_OperKeep.1) ,XIC(Sts_Maint) ]XIO(Sts_NotRdy)XIO(Wrk_Run)OTL(Wrk_Jog);
   // If the drive is being jogged, run the Jog Timer.
   39: XIC(Wrk_Jog)TON(Wrk_JogT,?,?);
   // If the drive is changed to a Mode other than Oper or Maint,
   // or if the Jog command goes away,
   // or if the Jog command does not clear within the Maximum Jog Time,
   // stop jogging.
   40: [[XIO(Sts_Oper) ,XIC(Cfg_ProgKeep.1) ] [XIO(Sts_Prog) ,XIO(Cfg_OperKeep.1) ] XIO(Sts_Maint) ,XIO(OCmd_Jog) ,XIC(Wrk_JogT.DN) NEQ(Wrk_JogT.PRE,0) ]OTU(Wrk_Jog);
